(* IEC 61131-3 sources: Industry-PLC-LLM/data/PLCBEAD_repo/PLCBEAD_PLCEmbed-main/PLC-BEAD/Source/GEB/CYCLE_4, 1 file *)

(* ---- CYCLE_4.ST ---- *)
FUNCTION_BLOCK T_PLC_MS_block
	VAR_OUTPUT
		T_PLC_MS :	UDINT;
	END_VAR

	VAR
		PLC_TICKS_PER_SEC :	INT;
		PLC_SYS_TICK_CNT :	DINT;
	END_VAR

	VAR
		debug :	BOOL;(*Debug-Mode ON / OFF*)
		N :	INT;(*Debug-Faktor*)
		Offset :	UDINT;(*Debug-Offset*)
		temp :	DWORD := DWORD#1;(*Debug-Offset*)
		MODE :	BOOL;(*modus*)
		faktor :	UDINT;(*Systemtakt-Faktor*)
		init :	BOOL;
		v_plc_ticks_per_sec :	UDINT;
		base :	UDINT := UDINT#1000;
	END_VAR

	IF init = FALSE THEN
		v_plc_ticks_per_sec := INT_TO_UDINT(PLC_TICKS_PER_SEC);
		IF v_plc_ticks_per_sec = UDINT#1024 THEN
			faktor := UDINT#1;
			MODE := FALSE;
		ELSIF v_plc_ticks_per_sec > UDINT#0 THEN
			IF v_plc_ticks_per_sec <= base THEN
				faktor := base / v_plc_ticks_per_sec;
				MODE := FALSE;
			ELSE
				faktor := v_plc_ticks_per_sec / base;
				MODE := TRUE;
			END_IF;
		ELSE
			faktor := UDINT#1;
		END_IF;
		init := TRUE;
	END_IF;

	IF MODE THEN
		T_PLC_MS := DINT_TO_UDINT(PLC_SYS_TICK_CNT) / faktor;
	ELSE
		T_PLC_MS := DINT_TO_UDINT(PLC_SYS_TICK_CNT) * faktor;
	END_IF;

	IF debug THEN
		T_PLC_MS := (DWORD_TO_UDINT(SHL(UDINT_TO_DWORD(T_PLC_MS),N) OR SHL(temp,N)) - UDINT#1) + Offset;
	END_IF;

END_FUNCTION_BLOCK

FUNCTION_BLOCK CYCLE_4

	VAR_INPUT
		E :	BOOL := TRUE;
		T0 :	TIME;
		T1 :	TIME;
		T2 :	TIME;
		T3 :	TIME;
		S0 :	BOOL;
		SX :	INT;
		SL :	BOOL;
	END_VAR

	VAR_OUTPUT
		STATE :	INT;
	END_VAR

	VAR
		TX :	TIME;
		last :	TIME;
		init :	BOOL;
		T_PLC_MS :	T_PLC_MS_block;
		SLL :	BOOL;
	END_VAR

	T_PLC_MS();
	TX:= UDINT_TO_TIME(T_PLC_MS.T_PLC_MS);

	(* init on fiRST cycle *)
	IF NOT init THEN
		init := TRUE;
		last := TX;
	END_IF;

	SLL := SL;
	IF E THEN
		IF SLL THEN
			(* when sx > 0 then the STATE sx is forced to START *)
			STATE:= LIMIT(0,SX,3);
			last := TX;
			(* this is to avoid to reset sx from the calling programm it does work fine on codesys but i am not sure abOUT other systems, becaUSE we are writing to an input *)
			SLL := FALSE;
		ELSE
			CASE STATE OF
				0 :	(* wait for T0 and switch to next cycle *)
					IF SUB_TIME(TX, last) >= T0 THEN
						STATE := 1;
						last := TX;
					END_IF;
				1 : (* wait for T1 over 1st cycle *)
					IF SUB_TIME(TX, last) >= T1 THEN
						STATE := 2;
						last := TX;
					END_IF;
				2 : (* wait for T1 over 1st cycle *)
					IF SUB_TIME(TX, last) >= T2 THEN
						STATE := 3;
						last := TX;
					END_IF;
				3 : (* wait for T2 over 2nd cycle *)
					IF SUB_TIME(TX, last) >= T3 THEN
						IF S0 THEN STATE := 0; END_IF; (* if S0 is false, the sequence STOPs at STATE 3 *)
						last := TX;
					END_IF;
			END_CASE;
		END_IF;
	ELSE
		STATE := 0;
		last := TX;
	END_IF;

END_FUNCTION_BLOCK

PROGRAM program0
  VAR
	E  :	BOOL ;
	T0 :	TIME;
	T1 :	TIME;
	T2 :	TIME;
	T3 :	TIME;
	S0 :	BOOL;
	SX :	INT;
	SL :	BOOL;

	STATE :	INT;

	func_block : CYCLE_4;
  END_VAR
	func_block.E   :=E ;
	func_block.T0  :=T0;
	func_block.T1  :=T1;
	func_block.T2  :=T2;
	func_block.T3  :=T3;
	func_block.S0  :=S0;
	func_block.SX  :=SX;
	func_block.SL  :=SL;
	func_block();
	STATE := func_block.STATE;
END_PROGRAM
